{attribute addProperty BoxType "EJ6224-0000-0016"}
{attribute addProperty Id "Device_DiagAT %I*BOOL8113Device_StateAT %I*BOOL8116"}
{attribute addProperty CRC "878559470"}
{attribute addProperty SizeInBites "16"}
{attribute addProperty SizeInBytes "2"}
TYPE DeviceState_Inputs_Device_345DC0EE :
STRUCT
	{attribute addProperty Name "Device_Diag"}
	Device_Diag AT %I* : BOOL;
	{attribute addProperty Name "Device_State"}
	Device_State AT %I* : BOOL;
END_STRUCT
END_TYPE

(* stored: Version 1.2.0.0, ProductVersion 3.1.4024.9
   DUT DeviceState_Inputs_Device_345DC0EE: Id {f48186e5-f8a7-41f4-aa12-4b699f9dd5cc} *)
